// TIA Portal project "2022.10.18_F_视觉分拣" (V17)

(* hardware
DEVICE "S7-1200 station_1"  S7-1200 Station
   slot 0: "Rack_0"  S7-1200 Rack  Rack  V1.0
   slot 1: "PLC_1"  CPU 1214C DC/DC/Rly  6ES7 214-1HG40-0XB0  V4.5
*)

// ===== PLC "PLC_1"  CPU 1214C DC/DC/Rly =====

VAR_GLOBAL   // PLC tag table "默认变量表"
   "启动" AT %I0.0 : Bool;
   "停止" AT %I0.1 : Bool;
   "复位" AT %I0.2 : Bool;
   "急停" AT %I0.3 : Bool;
   "左电传感器" AT %I0.5 : Bool;
   "右电传感器" AT %I0.6 : Bool;
   "直行传感器" AT %I0.7 : Bool;
   "手动模式" AT %I1.0 : Bool;
   "自动模式" AT %I1.1 : Bool;
   "启动指示灯" AT %Q0.0 : Bool;
   "停止指示灯" AT %Q0.1 : Bool;
   "复位指示灯" AT %Q0.2 : Bool;
   "进料输送机" AT %Q0.3 : Bool;
   "直行电机" AT %Q0.4 : Bool;
   "左换向" AT %Q0.5 : Bool;
   "右换向" AT %Q0.6 : Bool;
   "后1_原料输送机" AT %Q0.7 : Bool;
   "左1带_基座" AT %Q1.0 : Bool;
   "右1带_产品盖" AT %Q1.1 : Bool;
   "视觉相机数据" AT %ID30 : DWord;
   "生成物料" AT %Q1.2 : Bool;
   "停止挡板" AT %Q1.3 : Bool;
END_VAR

DATA_BLOCK "核心功能区DB"   // DB1
{ S7_Optimized_Access := 'TRUE' }
VERSION : 0.1
   VAR
      程序步 : Int;
      中间变量2 : Bool;
      中间变量1 : Bool;
      中间变量3 : Bool;
   END_VAR
BEGIN
END_DATA_BLOCK

ORGANIZATION_BLOCK "Main"   // OB1, LAD, ProgramCycle
TITLE = "Main Program Sweep (Cycle)"
{ S7_Optimized_Access := 'TRUE' }
VERSION : 0.1
   VAR_INPUT
      Initial_Call : Bool;   // Initial call of this OB
      Remanence : Bool;   // =True, if remanent data are available
   END_VAR
   VAR_TEMP   // added for the SCL form of the ladder/FBD networks
      _w1 : Bool;
   END_VAR
BEGIN

REGION Network 2: 实现产品物料判断
   // 1、4为产品原料  创建程序步
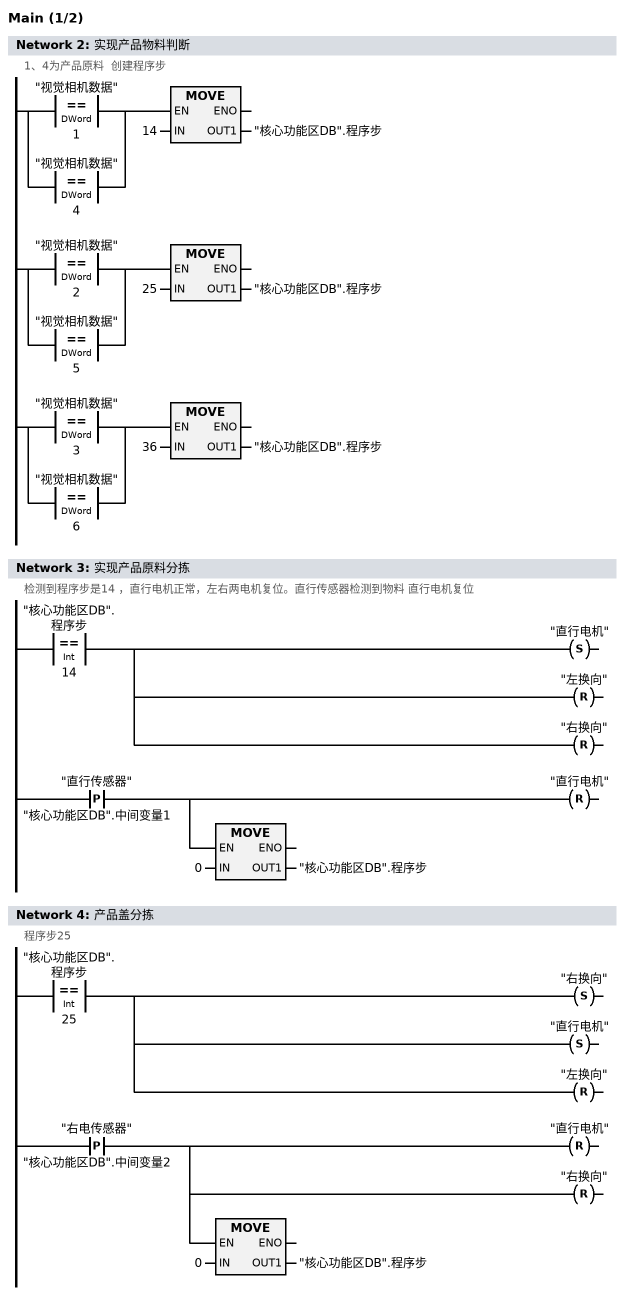
   RUNG wire#powerrail
      { S7_Templates := "SrcType := DWord" } EQ_Contact(in1 := "视觉相机数据", in2 := 1)
      wire#w1
      Move(in := 14, out1 => "核心功能区DB".程序步)
   END_RUNG
   RUNG wire#powerrail
      { S7_Templates := "SrcType := DWord" } EQ_Contact(in1 := "视觉相机数据", in2 := 4)
   END_RUNG wire#w1
   RUNG wire#powerrail
      { S7_Templates := "SrcType := DWord" } EQ_Contact(in1 := "视觉相机数据", in2 := 2)
      wire#w2
      Move(in := 25, out1 => "核心功能区DB".程序步)
   END_RUNG
   RUNG wire#powerrail
      { S7_Templates := "SrcType := DWord" } EQ_Contact(in1 := "视觉相机数据", in2 := 5)
   END_RUNG wire#w2
   RUNG wire#powerrail
      { S7_Templates := "SrcType := DWord" } EQ_Contact(in1 := "视觉相机数据", in2 := 3)
      wire#w3
      Move(in := 36, out1 => "核心功能区DB".程序步)
   END_RUNG
   RUNG wire#powerrail
      { S7_Templates := "SrcType := DWord" } EQ_Contact(in1 := "视觉相机数据", in2 := 6)
   END_RUNG wire#w3
   // the same network as SCL:
   IF ("视觉相机数据" = 1) OR ("视觉相机数据" = 4) THEN "核心功能区DB".程序步 := 14; END_IF;
   IF ("视觉相机数据" = 2) OR ("视觉相机数据" = 5) THEN "核心功能区DB".程序步 := 25; END_IF;
   IF ("视觉相机数据" = 3) OR ("视觉相机数据" = 6) THEN "核心功能区DB".程序步 := 36; END_IF;
END_REGION

REGION Network 3: 实现产品原料分拣
   // 检测到程序步是14 ，直行电机正常，左右两电机复位。直行传感器检测到物料 直行电机复位
   RUNG wire#powerrail
      { S7_Templates := "SrcType := Int" } EQ_Contact(in1 := "核心功能区DB".程序步, in2 := 14)
      wire#w1
      S_Coil( "直行电机" )
   END_RUNG
   RUNG wire#w1
      R_Coil( "左换向" )
   END_RUNG
   RUNG wire#w1
      R_Coil( "右换向" )
   END_RUNG
   RUNG wire#powerrail
      P_Contact(operand := "直行传感器", bit := "核心功能区DB".中间变量1)
      wire#w2
      R_Coil( "直行电机" )
   END_RUNG
   RUNG wire#w2
      Move(in := 0, out1 => "核心功能区DB".程序步)
   END_RUNG
   // the same network as SCL:
   IF "核心功能区DB".程序步 = 14 THEN
       "直行电机" := TRUE;
       "左换向" := FALSE;
       "右换向" := FALSE;
   END_IF;
   #_w1 := "直行传感器" AND NOT "核心功能区DB".中间变量1;   // rising edge of "直行传感器"
   "核心功能区DB".中间变量1 := "直行传感器";
   IF #_w1 THEN
       "直行电机" := FALSE;
       "核心功能区DB".程序步 := 0;
   END_IF;
END_REGION

REGION Network 4: 产品盖分拣
   // 程序步25
   RUNG wire#powerrail
      { S7_Templates := "SrcType := Int" } EQ_Contact(in1 := "核心功能区DB".程序步, in2 := 25)
      wire#w1
      S_Coil( "右换向" )
   END_RUNG
   RUNG wire#w1
      S_Coil( "直行电机" )
   END_RUNG
   RUNG wire#w1
      R_Coil( "左换向" )
   END_RUNG
   RUNG wire#powerrail
      P_Contact(operand := "右电传感器", bit := "核心功能区DB".中间变量2)
      wire#w2
      R_Coil( "直行电机" )
   END_RUNG
   RUNG wire#w2
      R_Coil( "右换向" )
   END_RUNG
   RUNG wire#w2
      Move(in := 0, out1 => "核心功能区DB".程序步)
   END_RUNG
   // the same network as SCL:
   IF "核心功能区DB".程序步 = 25 THEN
       "右换向" := TRUE;
       "直行电机" := TRUE;
       "左换向" := FALSE;
   END_IF;
   #_w1 := "右电传感器" AND NOT "核心功能区DB".中间变量2;   // rising edge of "右电传感器"
   "核心功能区DB".中间变量2 := "右电传感器";
   IF #_w1 THEN
       "直行电机" := FALSE;
       "右换向" := FALSE;
       "核心功能区DB".程序步 := 0;
   END_IF;
END_REGION

REGION Network 5: 产品基座分拣
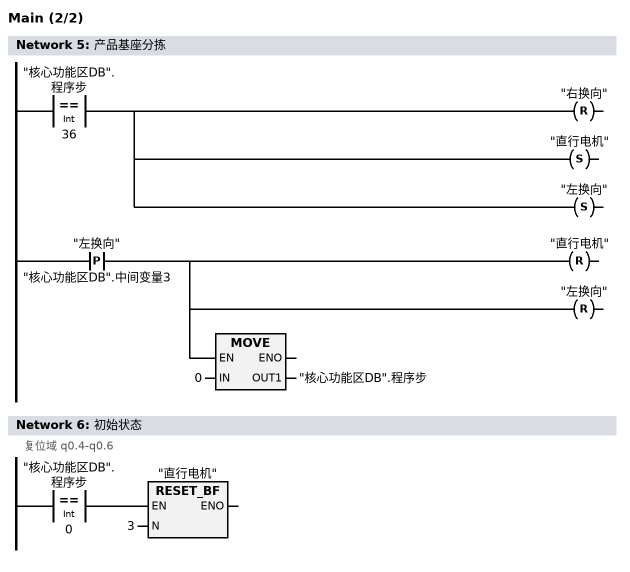
   RUNG wire#powerrail
      { S7_Templates := "SrcType := Int" } EQ_Contact(in1 := "核心功能区DB".程序步, in2 := 36)
      wire#w1
      R_Coil( "右换向" )
   END_RUNG
   RUNG wire#w1
      S_Coil( "直行电机" )
   END_RUNG
   RUNG wire#w1
      S_Coil( "左换向" )
   END_RUNG
   RUNG wire#powerrail
      P_Contact(operand := "左换向", bit := "核心功能区DB".中间变量3)
      wire#w2
      R_Coil( "直行电机" )
   END_RUNG
   RUNG wire#w2
      R_Coil( "左换向" )
   END_RUNG
   RUNG wire#w2
      Move(in := 0, out1 => "核心功能区DB".程序步)
   END_RUNG
   // the same network as SCL:
   IF "核心功能区DB".程序步 = 36 THEN
       "右换向" := FALSE;
       "直行电机" := TRUE;
       "左换向" := TRUE;
   END_IF;
   #_w1 := "左换向" AND NOT "核心功能区DB".中间变量3;   // rising edge of "左换向"
   "核心功能区DB".中间变量3 := "左换向";
   IF #_w1 THEN
       "直行电机" := FALSE;
       "左换向" := FALSE;
       "核心功能区DB".程序步 := 0;
   END_IF;
END_REGION

REGION Network 6: 初始状态
   // 复位域 q0.4-q0.6
   // no SCL statement known for RBitfield: written as a call
   IF "核心功能区DB".程序步 = 0 THEN RESET_BF(operand := "直行电机", n := 3); END_IF;
END_REGION
END_ORGANIZATION_BLOCK